FUNCTION_BLOCK ClearLinkMC EXTENDS FBA_Drive IMPLEMENTS I_EncodedDrive //I_PositionalDrive, I_ContinuousDrive
VAR_OUTPUT
	pulse AT %Q* : INT;
	brakeRelease AT %Q* : BOOL := TRUE;
	enable : BOOL;
	A : BOOL;
	B : BOOL;
	clear : BOOL;
END_VAR
VAR	
	outerLimit AT %I* : BOOL;
	hlfb AT %I* : REAL := -9999; //high level feedback, if -9999 then servo is idle
	
	outputRegister AT %Q* : INT;
	pulseRequest : INT;
	
	homingDelay : TON;
	resetPulse : TP;
	
	mode : (HOLD, TARGET, CONTINUOUS, RESET_ERR);
	calculation : (IDLE, DOWN, UP, CALCULATE, DONE);
	maxPosition : LREAL;
	
	position, targetPos : LREAL;
	
	pulsePosition : INT;
	pulseCounter : INT;
	rotationsPerPulse : INT; //revolutions per pulse
	displacementPerPulse : LREAL; //displacement per pulse
END_VAR
VAR_STAT CONSTANT
	resetWidth : TIME := T#500MS;
	delayWidth : TIME := T#500MS;
END_VAR
VAR //constructor
	homingDirection : BOOL; 			//homing direction - see <A>
	minPosition : LREAL;
	displacementPerRotation : LREAL; 	//displacement per revolution	
	unitsPerPulse : INT := 800; 		//800 Teknic units per rotation - default setting is 800 units (1 rotation) per pulse
END_VAR

//M-connector output register
outputRegister.0 := enable AND bEnable; 	//enable
outputRegister.1 := A; 						//direction bit
outputRegister.2 := B; 						//homing bit - after startup, set to TRUE to begin homing, then set to FALSE to finish homing
outputRegister.3 := clear; 					//reset bit

rotationsPerPulse := unitsPerPulse/800; //Teknic constant - 800 units per rotation
displacementPerPulse := displacementPerRotation * rotationsPerPulse;

resetPulse(IN:= , PT:= resetWidth, Q=> clear, ET=> ); //reset pulse

IF NOT enable AND NOT AtInnerLimit THEN
	homingComplete := FALSE;
	step := Homing.IDLE;
	mode := HOLD;
END_IF

override();

CASE mode OF		
	HOLD: //hold current position, no motion
		pulse := 0;
		pulseRequest := 0;
	
	TARGET:	//target a given position
		
		IF WithinTolerance(position, targetPos, displacementPerPulse) THEN
			pulseRequest := 0;
			pulse := 0;
			mode := HOLD;
			
		ELSIF NOT Active THEN
			A :=  position < targetPos;
			(*
			2 options to traverse to a target position:
				a)  send all pulses at once - single continuous motion but may exceed limits, check for bounds before setting
				b)  1 pulse at a time - choppy but safer
			*)
			pulseRequest := TO_INT(ABS(position - targetPos)/displacementPerPulse);
			//pulseRequest := 1;
		END_IF
		
	CONTINUOUS: //single pulses in the direction specified by moveContinuous()
		pulseRequest := 1;
		
	RESET_ERR: //reset pulse, servo may need to be rehomed aftewards
		pulse := 0;
		pulseRequest := 0;
		resetPulse.IN := TRUE;
		
		IF resetPulse.Q THEN
			resetPulse.IN := FALSE;
			mode := HOLD;
		END_IF
		
END_CASE

sequence();

PROPERTY Active : BOOL
GET
Active := hlfb <> -9999;
END_GET
END_PROPERTY

{attribute 'monitoring':='call'}
PROPERTY AtOuterLimit : BOOL
GET
AtOuterLimit := outerLimit <> limitSensorDefaultState;
END_GET
END_PROPERTY

METHOD PRIVATE calculatePositions : BOOL
(*
the purpose of this method is calculate the position at the outer limit

complete a full range traverse while counting the pulses, then multiply
	displacement per rotation
	rotations per pulse
	number of pulses for the traversal
and add to position at inner limit to get position at outer limit
*)
CASE calculation OF
	IDLE:
		calculation := DOWN;
		
	DOWN:
		moveContinuous(direction := MC_Negative_Direction);
		IF AtInnerLimit THEN
			calculation := UP;
			pulseCounter := 0;
		END_IF
		
	UP:
		moveContinuous(direction := MC_Positive_Direction);
		IF AtHome THEN
			maxPosition := minPosition + (displacementPerRotation * rotationsPerPulse * pulseCounter);
			calculation := DONE;
		END_IF
		
	DONE:
		calculation := 0;
		calculatePositions := TRUE;
		
END_CASE
END_METHOD

PROPERTY CurrentPosition : LREAL
GET
CurrentPosition := position;

//CurrentPosition := pulsePosition * displacementPerPulse;
END_GET
SET
position := CurrentPosition;
END_SET
END_PROPERTY

PROPERTY Error : BOOL
GET
END_GET
END_PROPERTY

METHOD homingSequence : BOOL
homingDelay(IN:= , PT:= delayWidth, Q=> , ET=> );

CASE step OF
	Homing.IDLE:
		enable := TRUE;
		A := FALSE;
		B := TRUE;
		brakeRelease := TRUE;
		
		homingComplete := FALSE;
		
		homingDelay.IN := TRUE;
		IF homingDelay.Q THEN
			homingDelay.IN := FALSE;
			//step := Homing.START;
			step := Homing.RETRY;
		END_IF
		
	Homing.START:
		IF homingDelay.Q THEN
			homingDelay.IN := FALSE;
			step := Homing.SET;
			
		ELSIF AtHome THEN
			homingDelay.IN := TRUE;
			
		ELSIF AtOuterLimit THEN
			step := Homing.RETRY;
		
		ELSE
			enable := TRUE;
			A := FALSE;
			B := TRUE;
			brakeRelease := TRUE;
		
		END_IF
	
	Homing.RETRY:
		IF AtInnerLimit THEN
			homingDelay.IN := TRUE;
			enable := FALSE;
			
			IF homingDelay.Q THEN
				homingDelay.IN := FALSE;
				step := Homing.START;
			END_IF
			
		ELSE
			enable := TRUE;
			A := FALSE;
			B := FALSE;
			brakeRelease := TRUE;
			
			mode := CONTINUOUS;
		END_IF

	Homing.SET:
		enable := TRUE;
		A := FALSE;
		B := FALSE;
		brakeRelease := TRUE;
		
		IF calculatePositions() THEN
			step := Homing.DONE;
		END_IF
		
	Homing.DONE:
		homingSequence := homingComplete := TRUE;
		
		pulsePosition := 0;
		
		mode := HOLD;
		step := Homing.IDLE;
	
END_CASE
END_METHOD

{attribute 'TcRpcEnable'}
METHOD moveAbsolute : BOOL
VAR_INPUT
	newTarget : LREAL;
END_VAR
IF target >= maxPosition AND target <= minPosition THEN
	A :=  position < targetPos;
	targetPos := newTarget;
	mode := TARGET;
	
	moveAbsolute := TRUE;
END_IF
END_METHOD

{attribute 'TcRpcEnable'}
METHOD moveContinuous : BOOL
VAR_INPUT
	direction : MC_Direction;
END_VAR
IF direction = MC_Negative_Direction THEN
	A := FALSE;
ELSIF direction = MC_Positive_Direction THEN
	A := TRUE;
END_IF

mode := CONTINUOUS;
END_METHOD

{attribute 'TcRpcEnable'}
METHOD moveRelative : BOOL
VAR_INPUT
	distance : LREAL;
END_VAR
targetPos := targetPos + distance;

mode := TARGET;
END_METHOD

METHOD PRIVATE override : BOOL
VAR_INPUT
END_VAR
(*
allowable motion is between AtHome and AtInnerLimit
*)
IF
	(AtHome AND A) OR
	(AtOuterLimit AND A) OR
	(AtInnerLimit AND NOT A)
THEN
	mode := HOLD;
END_IF

//--------------------

IF AtHome AND NOT Active THEN
	IF homingDirection THEN //homing is outwards
		position := maxPosition;
	ELSE
		position := minPosition;
	END_IF
	//pulsePosition := 0;

ELSIF AtInnerLimit AND NOT Active THEN
	IF homingDirection THEN //homing is outwards
		position := minPosition;
	ELSE
		position := maxPosition;
	END_IF
END_IF

(*
CASE mode OF		
	HOLD: //hold current position, no motion
		//
	
	TARGET:	//target a given position
		IF
			(AtHome AND TargetPosition > CurrentPosition) OR
			(AtOuterLimit AND TargetPosition > CurrentPosition) OR
			(AtInnerLimit AND TargetPosition < CurrentPosition)
		THEN
			mode := HOLD;
		END_IF
		
	CONTINUOUS: //single pulses in the direction specified by moveContinuous()
		IF
			(AtHome AND A) OR
			(AtOuterLimit AND A) OR
			(AtInnerLimit AND NOT A)
		THEN
			mode := HOLD;
		END_IF
		
	RESET_ERR: //reset pulse, servo may need to be rehomed aftewards
		//
		
END_CASE
*)
END_METHOD

METHOD reset : BOOL
VAR_INPUT
END_VAR
mode := RESET_ERR;
END_METHOD

METHOD PRIVATE sequence : BOOL
VAR_INPUT
END_VAR
IF Active THEN //servo is active
	IF A THEN //positive direction
		position := position + (displacementPerPulse * pulse);
		pulsePosition := pulsePosition + pulse;
		
		pulseCounter := pulseCounter + pulse;
	ELSE //negative direction
		position := position - (displacementPerPulse * pulse);
		pulsePosition := pulsePosition - pulse;
		
		pulseCounter := pulseCounter - pulse;
	END_IF
	pulse := 0; //pulses already received, can be set to 0 so position change is not compounded

ELSIF pulse = 0 THEN //servo is not active
	pulse := pulseRequest;
END_IF

pulseRequest := 0; //remove this if not working as intended
END_METHOD

METHOD stop : BOOL
VAR_INPUT
END_VAR
mode := HOLD;
END_METHOD

PROPERTY TargetPosition : LREAL
GET
END_GET
SET
targetPos := TargetPosition;
END_SET
END_PROPERTY

METHOD toHome : BOOL
VAR_INPUT
END_VAR
IF homingDirection THEN
	moveAbsolute(newTarget := maxPosition);
ELSE
	moveAbsolute(newTarget := minPosition);
END_IF
END_METHOD

END_FUNCTION_BLOCK

(* stored: Version 1.1.0.1, ProductVersion 3.1.4024.11
   POU ClearLinkMC: Id {82d395c8-897a-4c3b-989f-b99dc8146760}, SpecialFunc None
   Folder Private: Id {8d4dfb4b-1bc0-44fe-833d-9a6610663d13}
   Folder Properties: Id {d0779ed9-7013-4c4a-b5e7-14622eec869f}
   Property Active: Id {51689c1e-45ca-417f-9cf9-c85877f0bb33}
   Get Get: Id {1ba62c9f-3a34-481e-824a-0d65f3c6dff9}
   Property AtOuterLimit: Id {b968d47e-33dc-4e0f-b026-4fb76aa61d26}
   Get Get: Id {cd7ff1e2-65b0-4e28-b52f-2460f259be3e}
   Method calculatePositions: Id {93e72d7f-274c-4c53-979f-01532584dae3}
   Property CurrentPosition: Id {239591d6-8c9f-48a8-b8f2-e85872491b81}
   Get Get: Id {dc432c76-65d6-4e95-aa99-ce181ef2b386}
   Set Set: Id {d6f9c12b-1771-47bd-bf3a-b45d3c8818f2}
   Property Error: Id {6fbed130-ecef-45a8-a1d2-b4c51d85eca5}
   Get Get: Id {bfe6b58a-1695-41f1-9a43-74ca3f82e667}
   Method homingSequence: Id {ed7f9015-f217-4688-b191-db86d43e2b15}
   Method moveAbsolute: Id {dc77def1-bef9-43df-afd0-8ca352bd4ae2}
   Method moveContinuous: Id {56e37924-ed1f-434c-b8b5-86f83bcd5e14}
   Method moveRelative: Id {1770bae9-9ea8-4155-8a6e-b332d1abb598}
   Method override: Id {12f80332-3269-42b5-a267-e03e0f51e546}
   Method reset: Id {b78ab13d-678d-4b52-8830-ac5e90a85d68}
   Method sequence: Id {d3e76146-deb6-4a1c-bf00-057dae828590}
   Method stop: Id {b371037c-73c2-41cf-af60-cf703d5e079a}
   Property TargetPosition: Id {f459a582-972a-457c-9b48-2c8f2f4f4b42}
   Get Get: Id {229ed5b6-997e-4342-8be7-b4d85be1a8ce}
   Set Set: Id {957b0a36-861d-4a45-bc74-b57187f3168d}
   Method toHome: Id {3efa7aa4-d0b4-43df-9a67-d4c2edb36507} *)
